// TIA Portal V18 export
// export: Created 2026-06-12T02:00:00Z, ExportSetting WithDefaults
VAR_GLOBAL   // PLC tag table "PLC_AI_B5_Tags"
   AI_B5_CA_Fan_Motor_DE_Temp AT %MD400 : Real;   // TEMP 50-80 °C
   AI_B5_CA_Fan_Motor_NDE_Temp AT %MD404 : Real;   // TEMP 50-80 °C
   AI_B5_CA_Fan_DE_Temp AT %MD408 : Real;   // TEMP 50-80 °C
   AI_B5_CA_Fan_NDE_Temp AT %MD412 : Real;   // TEMP 50-80 °C
   AI_B5_CA_Fan_DE_Vib AT %MD416 : Real;   // COUNT 0-10 mm/s
   AI_B5_CA_Fan_NDE_Vib AT %MD420 : Real;   // COUNT 0-10 mm/s
   AI_B5_SP_700FN03 AT %MD424 : Real;   // FLOW 100-200 L/h
   AI_B5_SP_700HES01 AT %MD428 : Real;   // FLOW 100-200 L/h
   AI_B5_SP_700DA4 AT %MD432 : Real;   // FREQ 20-30 Hz
   AI_B5_SP_700DA6 AT %MD436 : Real;   // FREQ 20-30 Hz
   AI_B5_SP_700DA7 AT %MD440 : Real;   // FREQ 20-30 Hz
   AI_B5_SP_700FN2_DA1 AT %MD444 : Real;   // FREQ 20-30 Hz
   AI_B5_Sep_Motor_Top_Temp AT %MD448 : Real;   // TEMP 50-80 °C
   AI_B5_Sep_Bottom_Bear_Temp AT %MD452 : Real;   // TEMP 50-80 °C
   AI_B5_Trend_Val_1 AT %MD456 : Real;   // PERCENT 0-100 %
   AI_B5_Trend_Val_2 AT %MD460 : Real;   // PERCENT 0-100 %
   AI_B5_Trend_Val_3 AT %MD464 : Real;   // PERCENT 0-100 %
   AI_B5_700FN03_RPM AT %MD468 : Real;   // RPM 800-1200 RPM
   AI_B5_700HES01_Flow AT %MD472 : Real;   // FLOW 100-200 L/h
   AI_B5_700FN10_Speed AT %MD476 : Real;   // FREQ 20-30 Hz
   AI_B5_700CM01_Current AT %MD480 : Real;   // CURRENT 50-200 A
   AI_B5_Lub_Stop_Time AT %MD484 : Real;   // COUNT 0-300 Sec
   AI_B5_Main_Drive_ReHealth AT %MD488 : Real;   // COUNT 0-300 Sec
   AI_B5_CM_LRS_IN AT %MD492 : Real;   // TEMP 50-80 °C
   AI_B5_CM_LRS_OUT AT %MD496 : Real;   // TEMP 50-80 °C
   AI_B5_CM_Mill_Oil_Temp AT %MD500 : Real;   // TEMP 50-80 °C
   AI_B5_CM_OilTrun_BER_Temp AT %MD504 : Real;   // TEMP 50-80 °C
   AI_B5_CM_OilTrun_BER2_Temp AT %MD508 : Real;   // TEMP 50-80 °C
   AI_B5_CM_OilPinion_BER_Temp AT %MD512 : Real;   // TEMP 50-80 °C
   AI_B5_CM_GB_IL_Shaft_BER AT %MD516 : Real;   // TEMP 50-80 °C
   AI_B5_CM_Running_Hours AT %MD520 : Real;   // COUNT 0-8760 Hr
   AI_B5_CM_PS1_1_KG AT %MD524 : Real;   // PRESSURE 7-8 bar
   AI_B5_CM_PS1_2_KG AT %MD528 : Real;   // PRESSURE 7-8 bar
   AI_B5_NIBS_Value AT %MD532 : Real;   // CURRENT 50-200 A
   AI_B5_800DC1_Temp AT %MD536 : Real;   // TEMP 50-80 °C
   AI_B5_800DC2_Temp AT %MD540 : Real;   // TEMP 50-80 °C
   AI_B5_800FN1_Speed AT %MD544 : Real;   // FREQ 20-30 Hz
   AI_B5_800FN2_Speed AT %MD548 : Real;   // FREQ 20-30 Hz
   AI_B5_800YF1_Flow AT %MD552 : Real;   // FLOW 100-200 L/h
   AI_B5_800YF2_Flow AT %MD556 : Real;   // FLOW 100-200 L/h
   AI_B5_Silo1_Level_Bar1 AT %MD560 : Real;   // LEVEL 0-100 %
   AI_B5_Silo1_Level_Bar2 AT %MD564 : Real;   // LEVEL 0-100 %
   AI_B5_Silo2_Level_Bar1 AT %MD568 : Real;   // LEVEL 0-100 %
   AI_B5_Silo2_Level_Bar2 AT %MD572 : Real;   // LEVEL 0-100 %
   AI_B5_700FN01_Speed AT %MD576 : Real;   // FREQ 20-30 Hz
   AI_B5_700FN02_Speed AT %MD580 : Real;   // FREQ 20-30 Hz
   AI_B5_700AS07_Speed AT %MD584 : Real;   // FREQ 20-30 Hz
   AI_B5_700AS08_Flow AT %MD588 : Real;   // FLOW 100-200 L/h
   AI_B5_700FN09_Speed AT %MD592 : Real;   // FREQ 20-30 Hz
   AI_B5_700SFM01_Speed AT %MD596 : Real;   // FREQ 20-30 Hz
   AI_B5_700DA1_Flow AT %MD600 : Real;   // FLOW 100-200 L/h
   AI_B5_700DA4_Flow AT %MD604 : Real;   // FLOW 100-200 L/h
   AI_B5_700DA6_Temp AT %MD608 : Real;   // TEMP 50-80 °C
   AI_B5_700DA7_Temp AT %MD612 : Real;   // TEMP 50-80 °C
   AI_B5_700BL1_Load AT %MD616 : Real;   // CURRENT 50-200 A
   AI_B5_700BL2_Load AT %MD620 : Real;   // CURRENT 50-200 A
   AI_B5_700AS9_Flow AT %MD624 : Real;   // FLOW 100-200 L/h
   AI_B5_700FN13_Speed AT %MD628 : Real;   // FREQ 20-30 Hz
END_VAR
